// TwinCAT 3 PLC project BuildingBlocks
// Title: Building Blocks
// Company: Anker Andersen A/S
// Author: Benjamin Nielsen
// ProjectVersion: 1.0.0
// Description: Building blocks for process sub-elements
// ProgramVersion: 3.1.4026.1+972e9c44872ad038b353624a861fd7e3244e9f75
// libraries:
//   Tc2_Standard, * (Beckhoff Automation GmbH)
//   Tc2_System, * (Beckhoff Automation GmbH)
//   Tc2_TcpIp, * (Beckhoff Automation GmbH)
//   Tc2_Utilities, * (Beckhoff Automation GmbH)
// project tree:
//   / PlcTask.TcTTO
//   POUs/ FB_ClockPulsNumber.TcPOU, FB_ClockPulsOnOff.TcPOU, FB_RandomNumberGenerator.TcPOU, FB_TcpCommunication.TcPOU, MAIN.TcPOU
//   Version/ Global_Version.TcGVL
// real-time tasks:
//   TASK PlcTask: cycle T#10ms, priority 20, ADS port 350

CONFIGURATION BuildingBlocks
    RESOURCE PLC ON TwinCAT3
        TASK PlcTask(INTERVAL := T#10ms, PRIORITY := 20);
        PROGRAM MAIN WITH PlcTask : MAIN;
    END_RESOURCE
END_CONFIGURATION

// ---- Version/Global_Version.TcGVL
{attribute 'TcGenerated'}
{attribute 'no-analysis'}
{attribute 'linkalways'}
// This function has been automatically generated from the project information.
VAR_GLOBAL CONSTANT
	{attribute 'const_non_replaced'}
	stLibVersion_Building_Blocks : ST_LibVersion := (iMajor := 1, iMinor := 0, iBuild := 0, iRevision := 0, nFlags := 0, sVersion := '1.0.0');
END_VAR

// ---- POUs/MAIN.TcPOU
PROGRAM MAIN
VAR
END_VAR

END_PROGRAM

// ---- POUs/FB_ClockPulsNumber.TcPOU
FUNCTION_BLOCK FB_ClockPulsNumber
VAR_INPUT
	bTrig				:BOOL;					// On a rising edge, uiNo of puls are generated
	bStop				:BOOL;					// Stop and reset pulses
	uiNo				:UINT;					// Number of pulses to be generated when bTrig is set high
	tPulsLengthOn 		:TIME;
	tPulsLengthOff 		:TIME;
END_VAR
VAR_OUTPUT
	bPuls				:BOOL;					// Output puls
END_VAR
VAR
	osTrig				:R_TRIG;				// One shot trigger for start of pulses
	osPuls				:R_TRIG;				// One shot trigger for output puls
	uiCount				:UINT;					// Reset puls count
	fbStart				:SR;					// Set/Reset for reset to main zone.
	fbClockPulsOnOff 	:FB_ClockPulsOnOff;
END_VAR

osTrig(CLK:= bTrig, Q=> );

// Set start signal
fbStart(SET1:= osTrig.Q, RESET:= (uiCount > uiNo) OR bStop, Q1=> );

// Reset start signal
IF fbStart.RESET THEN
	uiCount := 0;
END_IF

// Generate clock puls
fbClockPulsOnOff(bEnable:= fbStart.Q1 AND NOT bStop, tPulsLengthOn := tPulsLengthOn, tPulsLengthOff:= tPulsLengthOff, bPuls=>);

// Count number of output pulses
osPuls(CLK:= fbClockPulsOnOff.bPuls, Q=> );
IF osPuls.Q THEN
	uiCount := uiCount + 1;
END_IF

// Set output puls
IF uiCount <= uiNo THEN
	bPuls := fbClockPulsOnOff.bPuls;
ELSE
	bPuls := FALSE;
END_IF

END_FUNCTION_BLOCK

// ---- POUs/FB_ClockPulsOnOff.TcPOU
FUNCTION_BLOCK FB_ClockPulsOnOff
VAR_INPUT
	bEnable				:BOOL;		// When TRUE a clock puls is generated. If set FALSE the bPuls output is always FALSE
	tPulsLengthOn		:TIME;		// Time for on 
	tPulsLengthOff		:TIME;		// Time for off	
END_VAR
VAR_OUTPUT
	bPuls				:BOOL;		// Clock Puls
END_VAR
VAR
	fbTimer1			:TON;		// Internal timer
	fbTimer2			:TON;		// Internal timer
	tHalfPuls			:TIME;
	bTimerOut			:BOOL;
END_VAR

IF bEnable THEN
	fbTimer1(IN:= NOT fbTimer2.Q , PT:= tPulsLengthOn, Q=>bTimerOut , ET=> );
	fbTimer2(IN:= fbTimer1.Q, PT:= tPulsLengthOff, Q=> , ET=> );
	// Start with postive edge when enabled
	bPuls := NOT bTimerOut;	
ELSE
	fbTimer1(IN:=FALSE);
	fbTimer2(IN:=FALSE);
	bPuls := FALSE;
END_IF

END_FUNCTION_BLOCK

// ---- POUs/FB_RandomNumberGenerator.TcPOU
FUNCTION_BLOCK FB_RandomNumberGenerator
VAR_INPUT
	bNewNumber		:BOOL;
	nMinNumber		:DINT;
	nMaxNumber		:DINT;
END_VAR
VAR_OUTPUT
	bDone			:BOOL;
	nRandomNumber	:DINT;
END_VAR
VAR
	fbSystemTime 		:NT_GetTime;
    timeAsTimeStruct	:TIMESTRUCT;
	osNewNumber			:R_TRIG;
	iStatus				:INT;
	nResult				:DINT;
	fDiv				:DINT;
	syncTimer	        :TON;
	bBusy         	    :BOOL;
    bError          	:BOOL;
END_VAR

//Get local time of windows
fbSystemTime(
	START:=syncTimer.Q,
	TMOUT:=DEFAULT_ADS_TIMEOUT,
	TIMESTR=>timeAsTimeStruct,
	BUSY=>bBusy,
	ERR=>bError);

syncTimer(IN:=NOT bBusy AND NOT bError, PT:=T#1MS);

IF nMinNumber < 1 THEN
	nMinNumber := 1;
END_IF

IF nResult < 1 THEN
	nResult := 1;
END_IF

//One shot
osNewNumber(CLK:=bNewNumber);

IF osNewNumber.Q THEN
	iStatus := 0;
END_IF

CASE iStatus OF 
	0:
		IF osNewNumber.Q THEN
			bDone := FALSE;
			nResult := 0;
			fDiv := nMaxNumber - nMinNumber;
			nResult := (timeAsTimeStruct.wMinute + timeAsTimeStruct.wSecond + timeAsTimeStruct.wMilliseconds) MOD (fDiv + 1);
			nResult := nResult + nMinNumber;
			iStatus := 10;
		END_IF
	10:
		bDone := TRUE;
		nRandomNumber := nResult;
END_CASE

END_FUNCTION_BLOCK

// ---- POUs/FB_TcpCommunication.TcPOU
FUNCTION_BLOCK FB_TcpCommunication
VAR_INPUT
	SocketHandler			:T_HSOCKET;						//Socket handler for connection
	sRemoteHost				:STRING;						//IP Address to connection
	nRemotePort				:UDINT;							//Port to connection	
END_VAR
VAR_OUTPUT
	aMessage				:ARRAY[0..50] OF T_MaxString;	//Array that contains the read message
END_VAR
VAR
	sReadString				:T_MaxString;					//Read string	
	aReadBytes				:ARRAY[0..1023] OF BYTE;		//Read bytes
	nWriteLen				:UDINT;							//Write length
	ReadComplete			:R_TRIG;						//Read complete
	tRefreshRead			:FB_ClockPulsOnOff;				//Refresh read time
	tRefreshWrite			:FB_ClockPulsOnOff;				//Refresh write time
	WriteSignal				:F_TRIG;						//Write signal
	iN						:UINT;							//Array incrementer
	rConnectedBusy			:F_TRIG;						//Falling edge of connection busy
END_VAR

METHOD M_ConnectRead : BOOL
VAR_INPUT
	bConnectRead			:BOOL;							//Connect/Open Read TCP
	bClear					:BOOL;							//Clear read and write
END_VAR
VAR_OUTPUT
	bConnectedRead			:BOOL;							//Connected to read socket
END_VAR
VAR
	fbConnect				:FB_SocketConnect;				//Connect to socket
	fbDisconnect			:FB_SocketClose;				//Close communication
END_VAR
//Connect to read
IF bConnectRead THEN
	
	//Disconnect write port 
	fbDisconnect(hSocket:=SocketHandler);
	

	//Connect read port
	fbConnect(
		sRemoteHost:=sRemoteHost,
		nRemotePort:=nRemotePort, 
		bExecute:=TRUE,
		tTimeout:=T#45S,
		hSocket=>SocketHandler);
END_IF

//Reset command
bConnectRead := FALSE;

rConnectedBusy(CLK:=fbConnect.bBusy);

IF rConnectedBusy.Q AND NOT fbConnect.bError THEN
	bConnectedRead := TRUE;
	//bConnectedWrite := FALSE;
END_IF
END_METHOD

METHOD M_ConnectWrite : BOOL
VAR_INPUT
	bConnectWrite			:BOOL;							//Connect/Open write TCP
END_VAR
VAR_OUTPUT
	bConnectedWrite			:BOOL;							//Connected to write socket
END_VAR
VAR
	fbConnect				:FB_SocketConnect;				//Connect to socket
	fbDisconnect			:FB_SocketClose;				//Close communication
END_VAR
//Connect to write
IF bConnectWrite THEN
	
	//Disconnect write port 
	fbDisconnect(hSocket:=SocketHandler);
	

	//Connect read port
	fbConnect(
		sRemoteHost:=sRemoteHost,
		nRemotePort:=nRemotePort, 
		bExecute:=TRUE,
		tTimeout:=T#45S,
		hSocket=>SocketHandler);
END_IF

//Reset command
bConnectWrite := FALSE;

rConnectedBusy(CLK:=fbConnect.bBusy);

IF rConnectedBusy.Q AND NOT fbConnect.bError THEN
	bConnectedWrite := TRUE;
	//bConnectedRead := FALSE;
END_IF
END_METHOD

METHOD M_ReadFrom : BOOL
VAR_INPUT
	nMessageBufferSize		:UDINT;							//Message read array buffer size
	bClear					:BOOL;							//Clear read and write
END_VAR
VAR
	fbRead					:FB_SocketReceive;				//Read from socket
END_VAR
IF M_ConnectRead.bConnectedRead THEN

	//Refresh read timer
	tRefreshRead(bEnable:=TRUE, tPulsLengthOn:=T#200MS, tPulsLengthOff:=T#200MS);
	
	fbRead(
		hSocket:=SocketHandler, 
		cbLen:=SIZEOF(aReadBytes),
		pDest:=ADR(aReadBytes),
		bExecute:=tRefreshRead.bPuls);
		
	ReadComplete(CLK:=fbRead.nRecBytes > 0);
	
	
	//If byte read, copy into string.
	IF ReadComplete.Q THEN
		MEMCPY(destAddr:=ADR(sReadString), srcAddr:=ADR(aReadBytes),n:=fbRead.nRecBytes);
		aMessage[iN] := sReadString;
		MEMSET(destAddr:=ADR(aReadBytes),fillByte:=0, n:=fbRead.nRecBytes);
		MEMSET(destAddr:=ADR(sReadString),fillByte:=0, n:=fbRead.nRecBytes);
		iN:=iN+1;
	END_IF
END_IF;


//Clear read and write
IF bClear THEN
	tRefreshRead(bEnable:=FALSE);
	MEMSET(destAddr:=ADR(aReadBytes),fillByte:=0, n:=fbRead.nRecBytes);
	MEMSET(destAddr:=ADR(sReadString),fillByte:=0, n:=fbRead.nRecBytes);
	
	FOR iN := 0 TO 50 DO 
		aMessage[iN] := '';
	END_FOR
	
	bClear := FALSE;
END_IF
END_METHOD

METHOD M_WriteTo : BOOL
VAR_INPUT
	sWriteString			:T_MaxString;					//Write string
END_VAR
VAR
	fbWrite					:FB_SocketSend;					//Write to socket
	aWriteBytes				:ARRAY[0..1023] OF BYTE;		//Write bytes

END_VAR
IF M_ConnectWrite.bConnectedWrite THEN	
	
	//Refresh read timer
	tRefreshWrite(bEnable:=TRUE, tPulsLengthOn:=T#200MS, tPulsLengthOff:=T#200MS);

	
	IF tRefreshWrite.bPuls THEN
		//Get length of string written
		nWriteLen := INT_TO_UDINT(LEN(STR:=sWriteString));
	
		//Copy string into array of bytes
		MEMCPY(destAddr:=ADR(aWriteBytes),srcAddr:=ADR(sWriteString),n:=nWriteLen);
		iN := iN + 1;
	END_IF
		
	//Write byte array to TCP server
	fbWrite(
		hSocket:=SocketHandler, 
		cbLen:=nWriteLen,
		pSrc:=ADR(aWriteBytes),
		bExecute:=tRefreshWrite.bPuls);
END_IF;
END_METHOD

END_FUNCTION_BLOCK
